FUNCTION_BLOCK ConveyorCTLMulticast (* Basic Function Block Type *)
  (* Standard: 61499-2 *)
  (* Version 0.2, 2003-12-04, JHC, Rockwell Automation, Renamed for better indexing. *)
  (* Version 0.1, 2002-11-05, JHC, Rockwell Automation, Corrected missing ST element in Algorithm REQ. *)
  (* Version 0.0, 2000-05-30, JHC, Rockwell Automation *)
  (* Compiler header: package fb.rt.cs725; *)
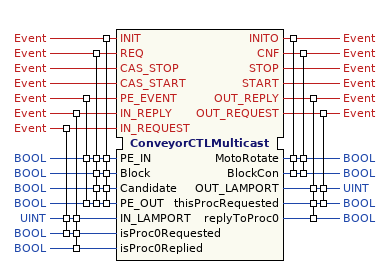
  EVENT_INPUT
    INIT WITH PE_IN, Block, Candidate, PE_OUT; (* Initialization Request *)
    REQ WITH PE_IN, Block, Candidate, PE_OUT; (* Normal Execution Request *)
    CAS_STOP;
    CAS_START;
    PE_EVENT WITH PE_OUT, PE_IN;
    IN_REPLY WITH IN_LAMPORT, isProc0Requested, isProc0Replied;
    IN_REQUEST WITH IN_LAMPORT, isProc0Requested;
  END_EVENT
  EVENT_OUTPUT
    INITO WITH MotoRotate, BlockCon; (* Initialization Confirm *)
    CNF WITH MotoRotate, BlockCon; (* Execution Confirmation *)
    STOP;
    START;
    OUT_REPLY WITH OUT_LAMPORT, thisProcRequested, replyToProc0;
    OUT_REQUEST WITH OUT_LAMPORT, thisProcRequested;
  END_EVENT
  VAR_INPUT
    PE_IN : BOOL; (* Input event qualifier *)
    Block : BOOL;
    Candidate : BOOL;
    PE_OUT : BOOL;
    IN_LAMPORT : UINT;
    isProc0Requested : BOOL;
    isProc0Replied : BOOL;
  END_VAR
  VAR_OUTPUT
    MotoRotate : BOOL; (* Output event qualifier *)
    BlockCon : BOOL;
    OUT_LAMPORT : UINT;
    thisProcRequested : BOOL;
    replyToProc0 : BOOL;
  END_VAR
  VAR
    lastPE : BOOL := 1;
    lastBlock : BOOL := 0;
    lamportTime : UINT;
    previousState : INT;
    allReplied : BOOL;
    replies : ARRAY [0..0] OF BOOL;
    requests : ARRAY [0..0] OF BOOL;
    I : INT;
  END_VAR
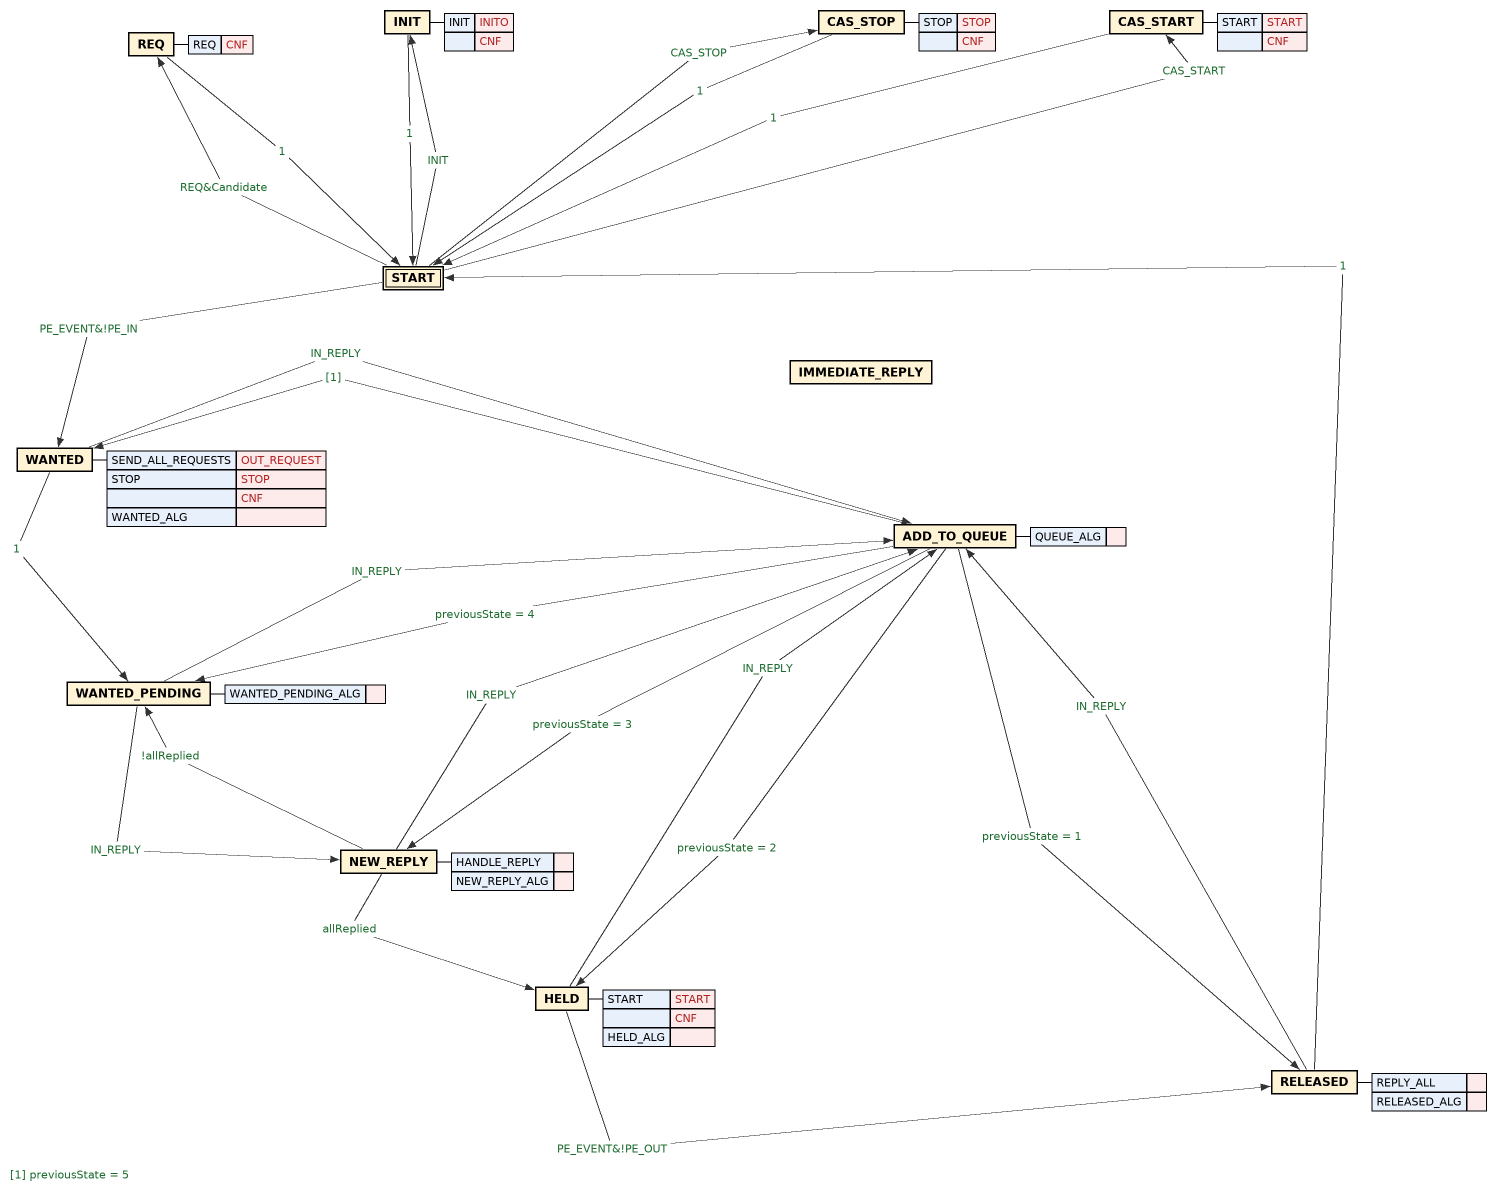
  EC_STATES
    START; (* Initial State *)
    INIT : INIT -> INITO, -> CNF; (* Initialization *)
    REQ : REQ -> CNF; (* Normal execution *)
    CAS_START : START -> START, -> CNF;
    CAS_STOP : STOP -> STOP, -> CNF;
    WANTED : SEND_ALL_REQUESTS -> OUT_REQUEST, STOP -> STOP, -> CNF, WANTED_ALG;
    HELD : START -> START, -> CNF, HELD_ALG;
    RELEASED : REPLY_ALL, RELEASED_ALG;
    WANTED_PENDING : WANTED_PENDING_ALG;
    NEW_REPLY : HANDLE_REPLY, NEW_REPLY_ALG;
    ADD_TO_QUEUE : QUEUE_ALG;
    IMMEDIATE_REPLY;
  END_STATES
  EC_TRANSITIONS
    START TO INIT := INIT;
    INIT TO START := 1;
    START TO REQ := REQ&Candidate;
    REQ TO START := 1;
    START TO CAS_START := CAS_START;
    CAS_START TO START := 1;
    START TO CAS_STOP := CAS_STOP;
    CAS_STOP TO START := 1;
    START TO WANTED := PE_EVENT&!PE_IN;
    WANTED TO WANTED_PENDING := 1;
    WANTED_PENDING TO NEW_REPLY := IN_REPLY;
    HELD TO RELEASED := PE_EVENT&!PE_OUT;
    NEW_REPLY TO WANTED_PENDING := !allReplied;
    NEW_REPLY TO HELD := allReplied;
    RELEASED TO START := 1;
    RELEASED TO ADD_TO_QUEUE := IN_REPLY;
    HELD TO ADD_TO_QUEUE := IN_REPLY;
    WANTED_PENDING TO ADD_TO_QUEUE := IN_REPLY;
    WANTED TO ADD_TO_QUEUE := IN_REPLY;
    NEW_REPLY TO ADD_TO_QUEUE := IN_REPLY;
    ADD_TO_QUEUE TO RELEASED := previousState = 1;
    ADD_TO_QUEUE TO HELD := previousState = 2;
    ADD_TO_QUEUE TO NEW_REPLY := previousState = 3;
    ADD_TO_QUEUE TO WANTED_PENDING := previousState = 4;
    ADD_TO_QUEUE TO WANTED := previousState = 5;
  END_TRANSITIONS
  ALGORITHM INIT IN ST: (* Initialization algorithm *)
MotoRotate := TRUE;
Block := FALSE;

System.out.println(this + " " + MotoRotate);
System.out.println(MotoRotate);

lamportTime := 0;
  END_ALGORITHM
  ALGORITHM REQ IN ST: (* Normally executed algorithm *)
//System.out.println(this +  " -> Candidate" + Candidate);
IF Candidate THEN
IF lastPE !:= PE_IN THEN
IF NOT PE_IN THEN
BlockCon:= TRUE;
System.out.println("BlockCon = true");
ELSE
BlockCon:=FALSE;
System.out.println("BlockCon = false");
END_IF
lastPE := PE_IN;
END_IF
IF lastBlock !:= Block THEN
IF Block THEN
STOP.serviceEvent(this);
MotoRotate := FALSE;
System.out.println("Cas Stop");
ELSE
START.serviceEvent(this);
MotoRotate := TRUE;
System.out.println("Cas Start");
END_IF
lastBlock := Block;
END_IF
END_IF
  END_ALGORITHM
  ALGORITHM START IN ST:
MotoRotate:=TRUE;
System.out.println(this + " Start " + MotoRotate);

System.out.println("Start " + MotoRotate);
  END_ALGORITHM
  ALGORITHM STOP IN ST:
MotoRotate := FALSE;
System.out.println(this + " Stop " + MotoRotate);

System.out.println("Stop " + MotoRotate);
  END_ALGORITHM
  ALGORITHM SEND_ALL_REQUESTS IN ST:
OUT_LAMPORT := lamportTime;
thisProcRequested := TRUE;
  END_ALGORITHM
  ALGORITHM HANDLE_REPLY IN ST:
//first, check which processes are replying
IF (isProc0Replied = TRUE) THEN
    replies[0] := TRUE;
END_IF;

//now, check if all replies are present
allReplied := TRUE;
FOR I := 0 TO 0 DO
    IF replies[I] = FALSE THEN
        allReplied := FALSE;
    END_IF;
END_FOR
  END_ALGORITHM
  ALGORITHM REPLY_ALL IN ST:

  END_ALGORITHM
  ALGORITHM WANTED_PENDING_ALG IN ST:
previousState := 4;
  END_ALGORITHM
  ALGORITHM WANTED_ALG IN ST:
previousState := 5;
  END_ALGORITHM
  ALGORITHM NEW_REPLY_ALG IN ST:
previousState := 3;
  END_ALGORITHM
  ALGORITHM RELEASED_ALG IN ST:
previousState := 1;
  END_ALGORITHM
  ALGORITHM HELD_ALG IN ST:
previousState := 2;
  END_ALGORITHM
  ALGORITHM QUEUE_ALG IN ST:

  END_ALGORITHM
END_FUNCTION_BLOCK
